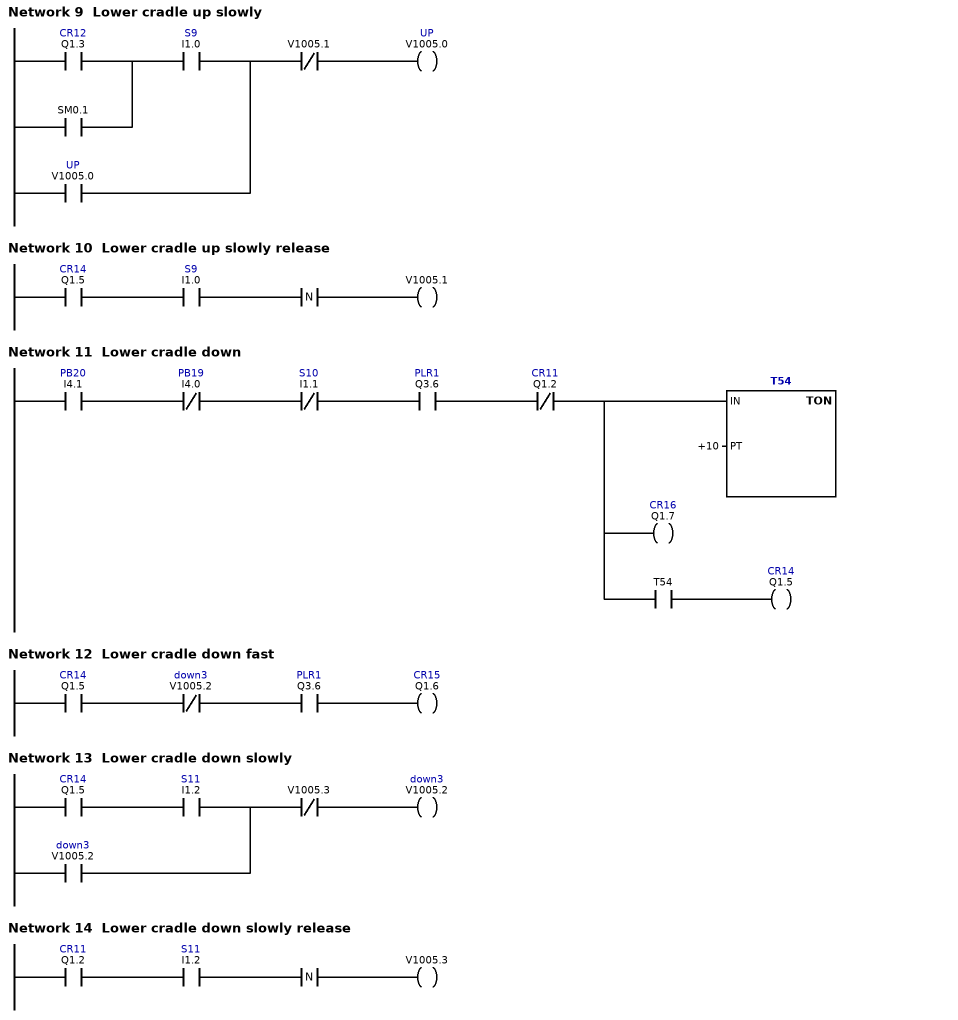
[picture p24: SBR7 networks 9-14]
Network 9 // Lower cradle up slowly
LD     CR12:Q1.3
O      SM0.1
A      S9:I1.0
O      UP:V1005.0
AN     V1005.1
=      UP:V1005.0
Network 10 // Lower cradle up slowly release
LD     CR14:Q1.5
A      S9:I1.0
ED
=      V1005.1
Network 11 // Lower cradle down
LD     PB20:I4.1
AN     PB19:I4.0
AN     S10:I1.1
A      PLR1:Q3.6
AN     CR11:Q1.2
TON    T54, +10
=      CR16:Q1.7
A      T54
=      CR14:Q1.5
Network 12 // Lower cradle down fast
LD     CR14:Q1.5
AN     down3:V1005.2
A      PLR1:Q3.6
=      CR15:Q1.6
Network 13 // Lower cradle down slowly
LD     CR14:Q1.5
A      S11:I1.2
O      down3:V1005.2
AN     V1005.3
=      down3:V1005.2
Network 14 // Lower cradle down slowly release
LD     CR11:Q1.2
A      S11:I1.2
ED
=      V1005.3
END_SUBROUTINE_BLOCK

SUBROUTINE_BLOCK Sheed_lead:SBR8
TITLE= SUBROUTINE COMMENTS
// Press F1 for help and example program 
BEGIN
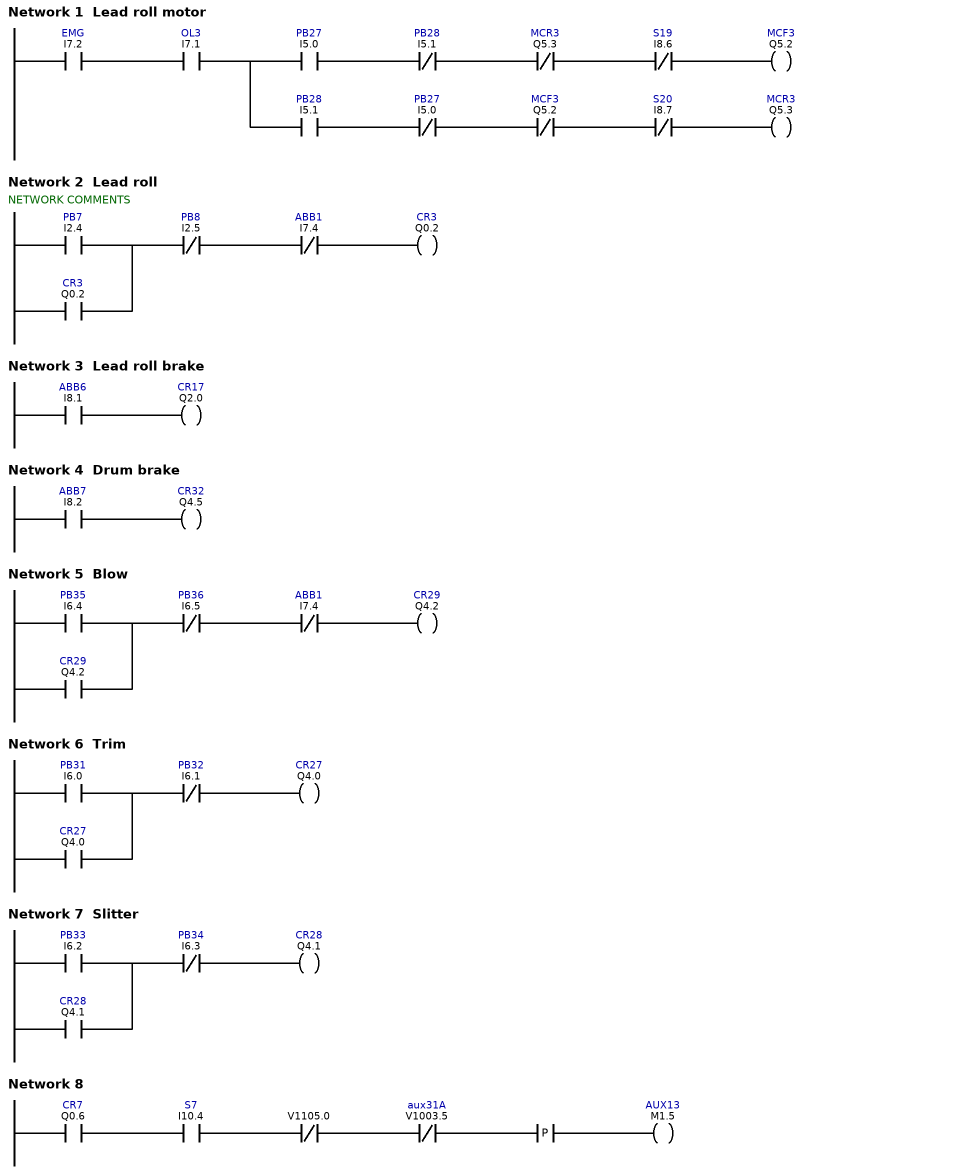
Network 1 // Lead roll motor
LD     EMG:I7.2
A      OL3:I7.1
LPS
A      PB27:I5.0
AN     PB28:I5.1
AN     MCR3:Q5.3
AN     S19:I8.6
=      MCF3:Q5.2
LPP
A      PB28:I5.1
AN     PB27:I5.0
AN     MCF3:Q5.2
AN     S20:I8.7
=      MCR3:Q5.3
Network 2 // Lead roll
//  NETWORK COMMENTS
LD     PB7:I2.4
O      CR3:Q0.2
AN     PB8:I2.5
AN     ABB1:I7.4
=      CR3:Q0.2
Network 3 // Lead roll brake
LD     ABB6:I8.1
=      CR17:Q2.0
Network 4 // Drum brake
LD     ABB7:I8.2
=      CR32:Q4.5
Network 5 // Blow
LD     PB35:I6.4
O      CR29:Q4.2
AN     PB36:I6.5
AN     ABB1:I7.4
=      CR29:Q4.2
Network 6 // Trim 
LD     PB31:I6.0
O      CR27:Q4.0
AN     PB32:I6.1
=      CR27:Q4.0
Network 7 // Slitter
LD     PB33:I6.2
O      CR28:Q4.1
AN     PB34:I6.3
=      CR28:Q4.1
Network 8
LD     CR7:Q0.6
A      S7:I10.4
AN     V1105.0
AN     aux31A:V1003.5
EU
=      AUX13:M1.5
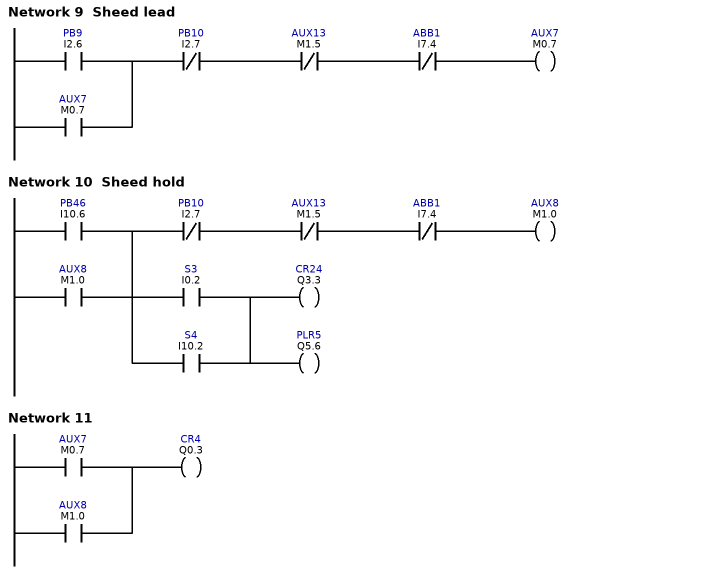
Network 9 // Sheed lead
LD     PB9:I2.6
O      AUX7:M0.7
AN     PB10:I2.7
AN     AUX13:M1.5
AN     ABB1:I7.4
=      AUX7:M0.7
Network 10 // Sheed hold
LD     PB46:I10.6
O      AUX8:M1.0
LPS
AN     PB10:I2.7
AN     AUX13:M1.5
AN     ABB1:I7.4
=      AUX8:M1.0
LPP
LD     S3:I0.2
O      S4:I10.2
ALD
=      CR24:Q3.3
=      PLR5:Q5.6
Network 11
LD     AUX7:M0.7
O      AUX8:M1.0
=      CR4:Q0.3
END_SUBROUTINE_BLOCK

SUBROUTINE_BLOCK Core_Chuck:SBR9
TITLE= 
// SUBROUTINE COMMENTS
// Press F1 for help and example program
//  
BEGIN
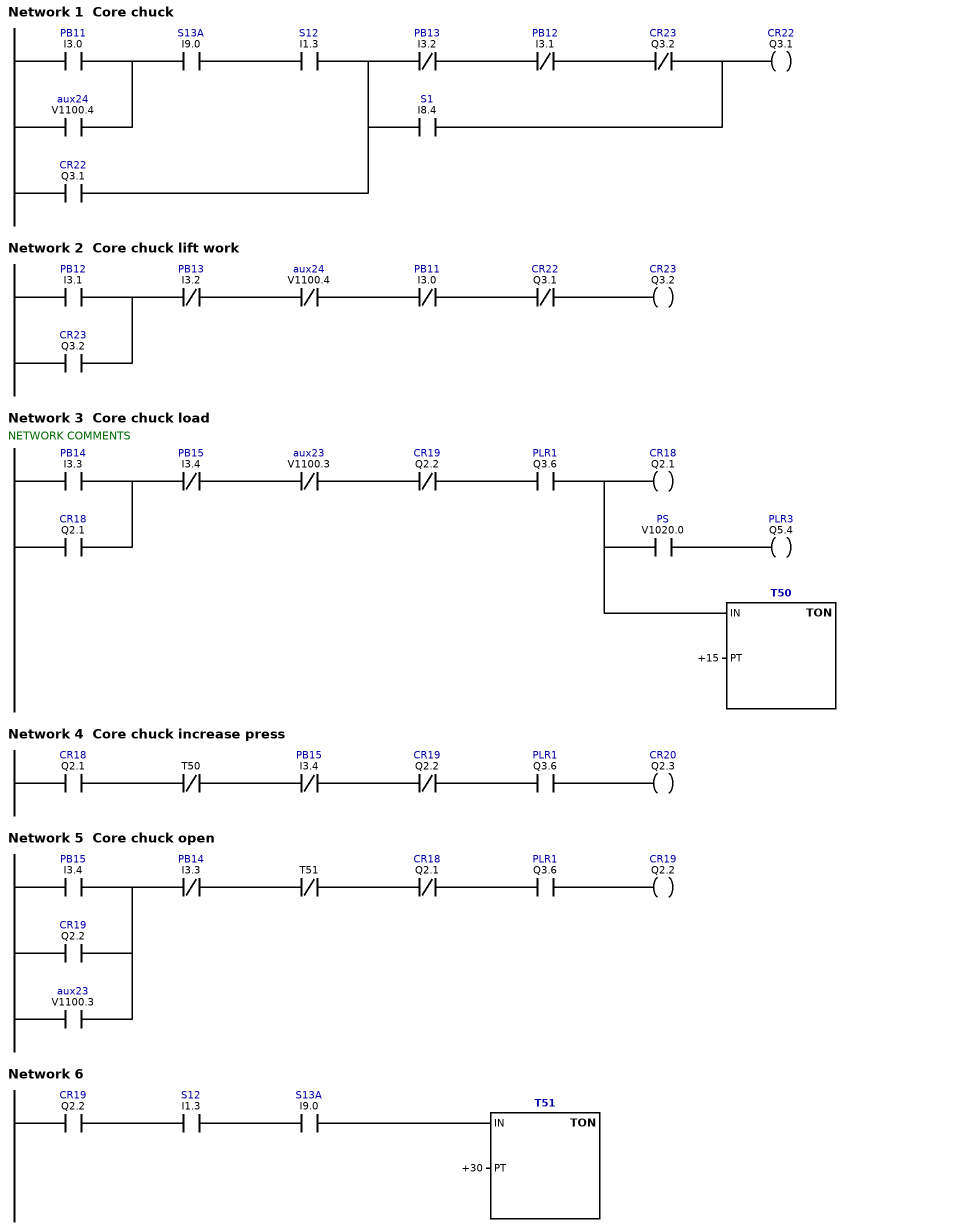
Network 1 // Core chuck
// 
// 
LD     PB11:I3.0
O      aux24:V1100.4
A      S13A:I9.0
A      S12:I1.3
O      CR22:Q3.1
LDN    PB13:I3.2
AN     PB12:I3.1
AN     CR23:Q3.2
O      S1:I8.4
ALD
=      CR22:Q3.1
Network 2 // Core chuck lift work
// 
// 
LD     PB12:I3.1
O      CR23:Q3.2
AN     PB13:I3.2
AN     aux24:V1100.4
AN     PB11:I3.0
AN     CR22:Q3.1
=      CR23:Q3.2
Network 3 // Core chuck load
//  NETWORK COMMENTS
LD     PB14:I3.3
O      CR18:Q2.1
AN     PB15:I3.4
AN     aux23:V1100.3
AN     CR19:Q2.2
A      PLR1:Q3.6
LPS
=      CR18:Q2.1
A      PS:V1020.0
=      PLR3:Q5.4
LPP
TON    T50, +15
Network 4 // Core chuck increase press
LD     CR18:Q2.1
AN     T50
AN     PB15:I3.4
AN     CR19:Q2.2
A      PLR1:Q3.6
=      CR20:Q2.3
Network 5 // Core chuck open
LD     PB15:I3.4
O      CR19:Q2.2
O      aux23:V1100.3
AN     PB14:I3.3
AN     T51
AN     CR18:Q2.1
A      PLR1:Q3.6
=      CR19:Q2.2
Network 6
LD     CR19:Q2.2
A      S12:I1.3
A      S13A:I9.0
TON    T51, +30
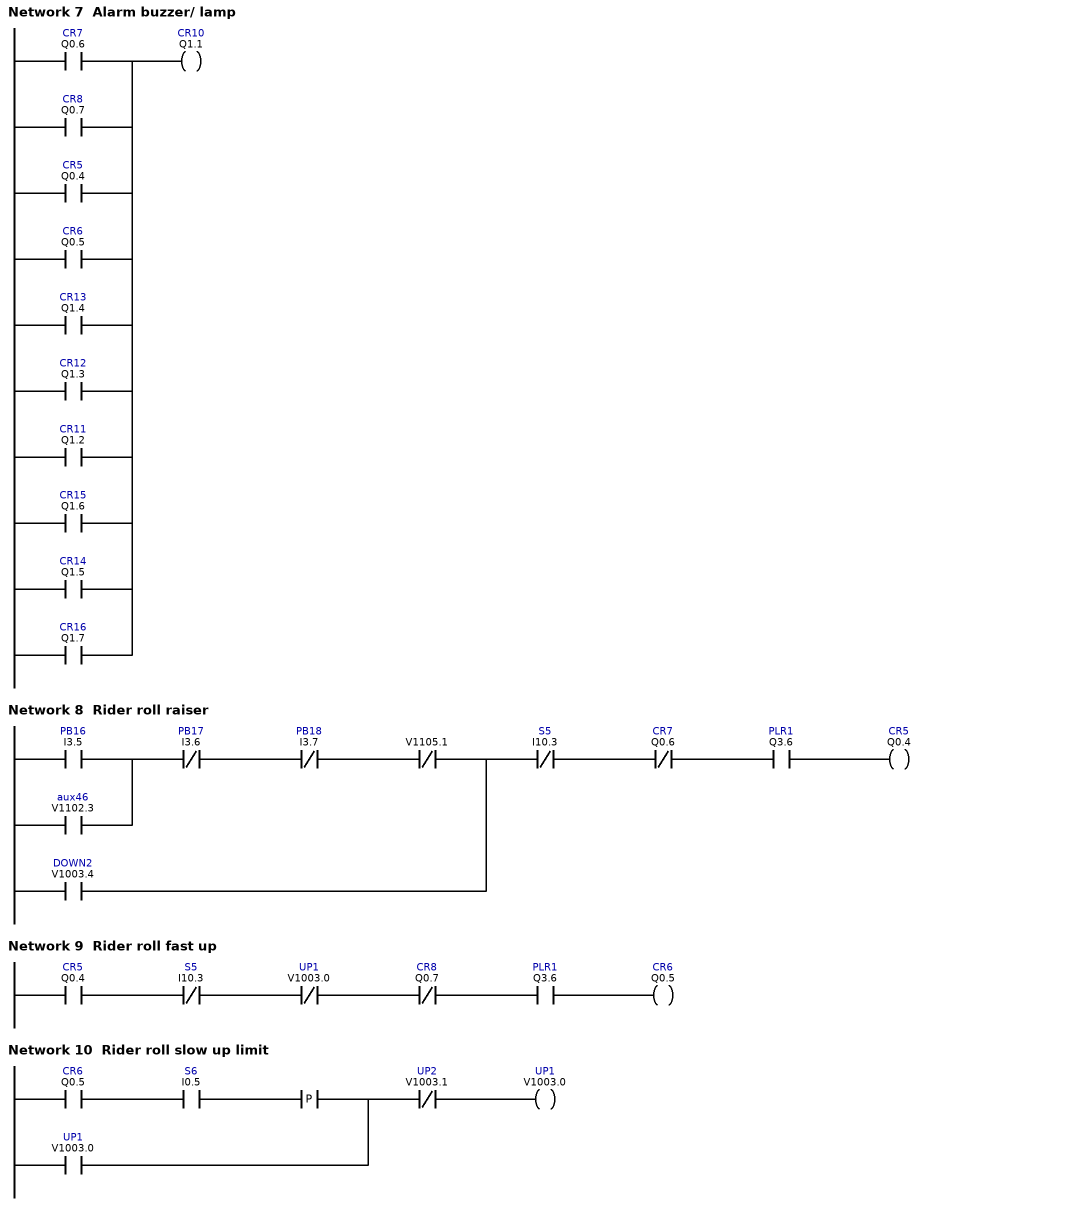
Network 7 // Alarm buzzer/ lamp
LD     CR7:Q0.6
O      CR8:Q0.7
O      CR5:Q0.4
O      CR6:Q0.5
O      CR13:Q1.4
O      CR12:Q1.3
O      CR11:Q1.2
O      CR15:Q1.6
O      CR14:Q1.5
O      CR16:Q1.7
=      CR10:Q1.1
Network 8 // Rider roll raiser
LD     PB16:I3.5
O      aux46:V1102.3
AN     PB17:I3.6
AN     PB18:I3.7
AN     V1105.1
O      DOWN2:V1003.4
AN     S5:I10.3
AN     CR7:Q0.6
A      PLR1:Q3.6
=      CR5:Q0.4
Network 9 // Rider roll fast up
LD     CR5:Q0.4
AN     S5:I10.3
AN     UP1:V1003.0
AN     CR8:Q0.7
A      PLR1:Q3.6
=      CR6:Q0.5
Network 10 // Rider roll slow up limit
LD     CR6:Q0.5
A      S6:I0.5
EU
O      UP1:V1003.0
AN     UP2:V1003.1
=      UP1:V1003.0
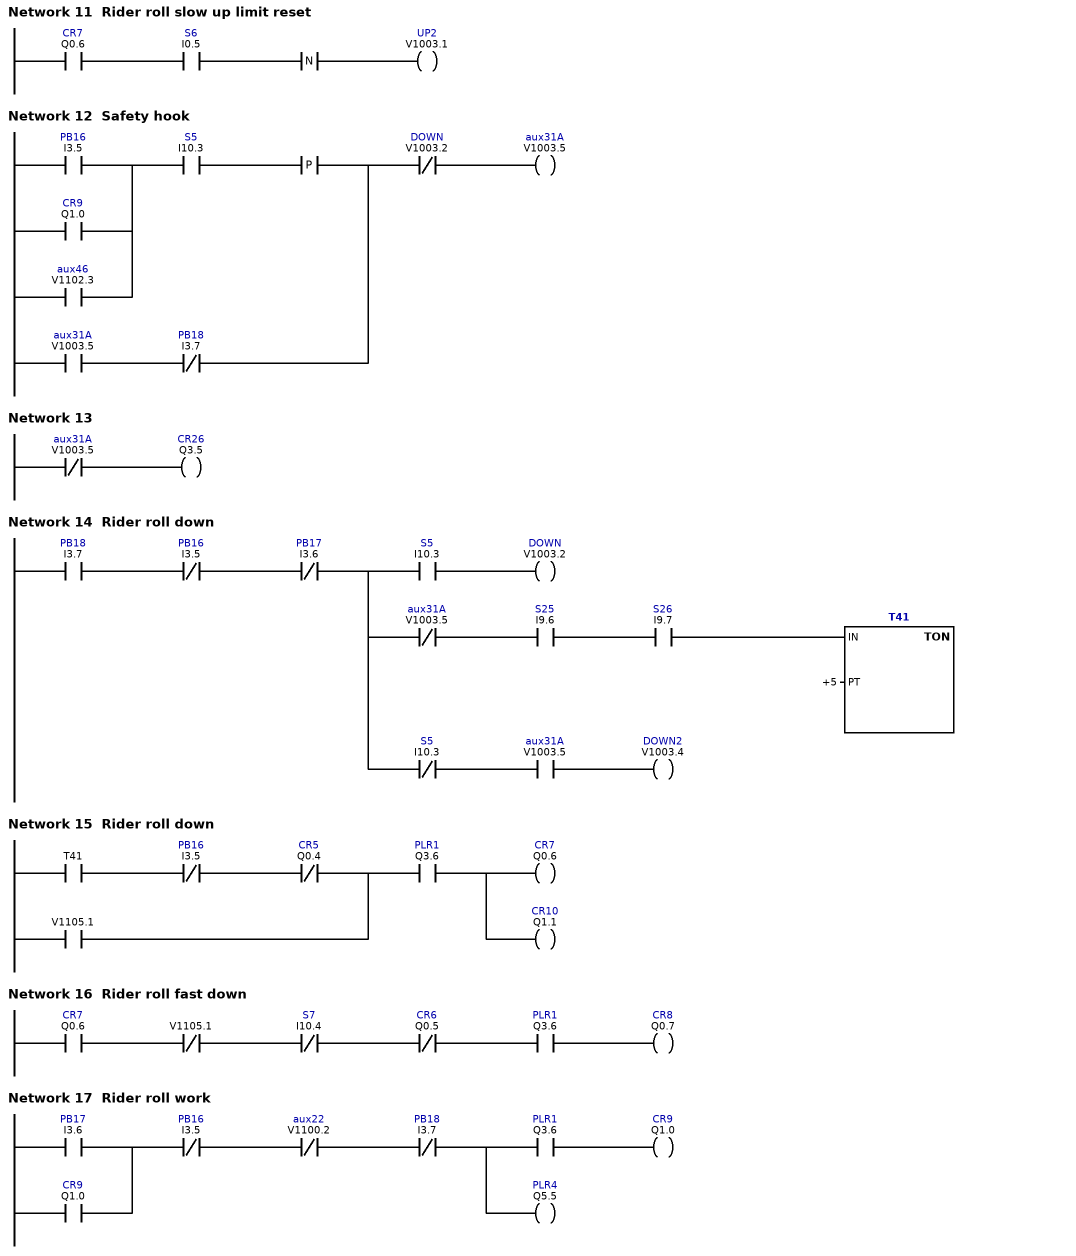
Network 11 // Rider roll slow up limit reset
LD     CR7:Q0.6
A      S6:I0.5
ED
=      UP2:V1003.1
Network 12 // Safety hook
LD     PB16:I3.5
O      CR9:Q1.0
O      aux46:V1102.3
A      S5:I10.3
EU
LD     aux31A:V1003.5
AN     PB18:I3.7
OLD
AN     DOWN:V1003.2
=      aux31A:V1003.5
Network 13
LDN    aux31A:V1003.5
=      CR26:Q3.5
Network 14 // Rider roll down
LD     PB18:I3.7
AN     PB16:I3.5
AN     PB17:I3.6
LPS
A      S5:I10.3
=      DOWN:V1003.2
LRD
AN     aux31A:V1003.5
A      S25:I9.6
A      S26:I9.7
TON    T41, +5
LPP
AN     S5:I10.3
A      aux31A:V1003.5
=      DOWN2:V1003.4
Network 15 // Rider roll down
LD     T41
AN     PB16:I3.5
AN     CR5:Q0.4
O      V1105.1
A      PLR1:Q3.6
=      CR7:Q0.6
=      CR10:Q1.1
Network 16 // Rider roll fast down
LD     CR7:Q0.6
AN     V1105.1
AN     S7:I10.4
AN     CR6:Q0.5
A      PLR1:Q3.6
=      CR8:Q0.7
Network 17 // Rider roll work
LD     PB17:I3.6
O      CR9:Q1.0
AN     PB16:I3.5
AN     aux22:V1100.2
AN     PB18:I3.7
LPS
A      PLR1:Q3.6
=      CR9:Q1.0
LPP
=      PLR4:Q5.5
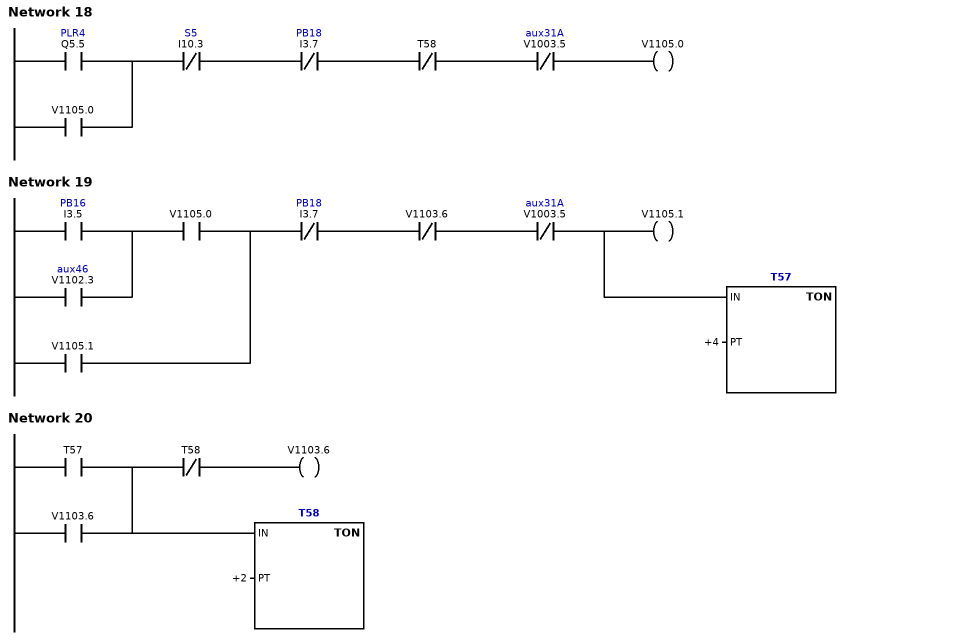
Network 18
LD     PLR4:Q5.5
O      V1105.0
AN     S5:I10.3
AN     PB18:I3.7
AN     T58
AN     aux31A:V1003.5
=      V1105.0
Network 19
LD     PB16:I3.5
O      aux46:V1102.3
A      V1105.0
O      V1105.1
AN     PB18:I3.7
AN     V1103.6
AN     aux31A:V1003.5
=      V1105.1
TON    T57, +4
Network 20
LD     T57
O      V1103.6
LPS
AN     T58
=      V1103.6
LPP
TON    T58, +2
END_SUBROUTINE_BLOCK

SUBROUTINE_BLOCK Value_1:SBR10
TITLE= SUBROUTINE COMMENTS
// Press F1 for help and example program 
VAR_INPUT
d1:REAL;	// LD0 
H:REAL;	// LD4 
END_VAR
VAR_OUTPUT
D:REAL;	// LD8 
END_VAR
VAR
TEMP1:REAL;	// LD12 
TEMP2:REAL;	// LD16 
TEMP3:REAL;	// LD20 
TEMP4:REAL;	// LD24 
TEMP5:REAL;	// LD28 
TEMP6:REAL;	// LD32 
TEMP7:REAL;	// LD36 
TEMP8:REAL;	// LD40 
TEMP9:REAL;	// LD44 
TEMP10:REAL;	// LD48 
TEMP11:REAL;	// LD52 
END_VAR
BEGIN
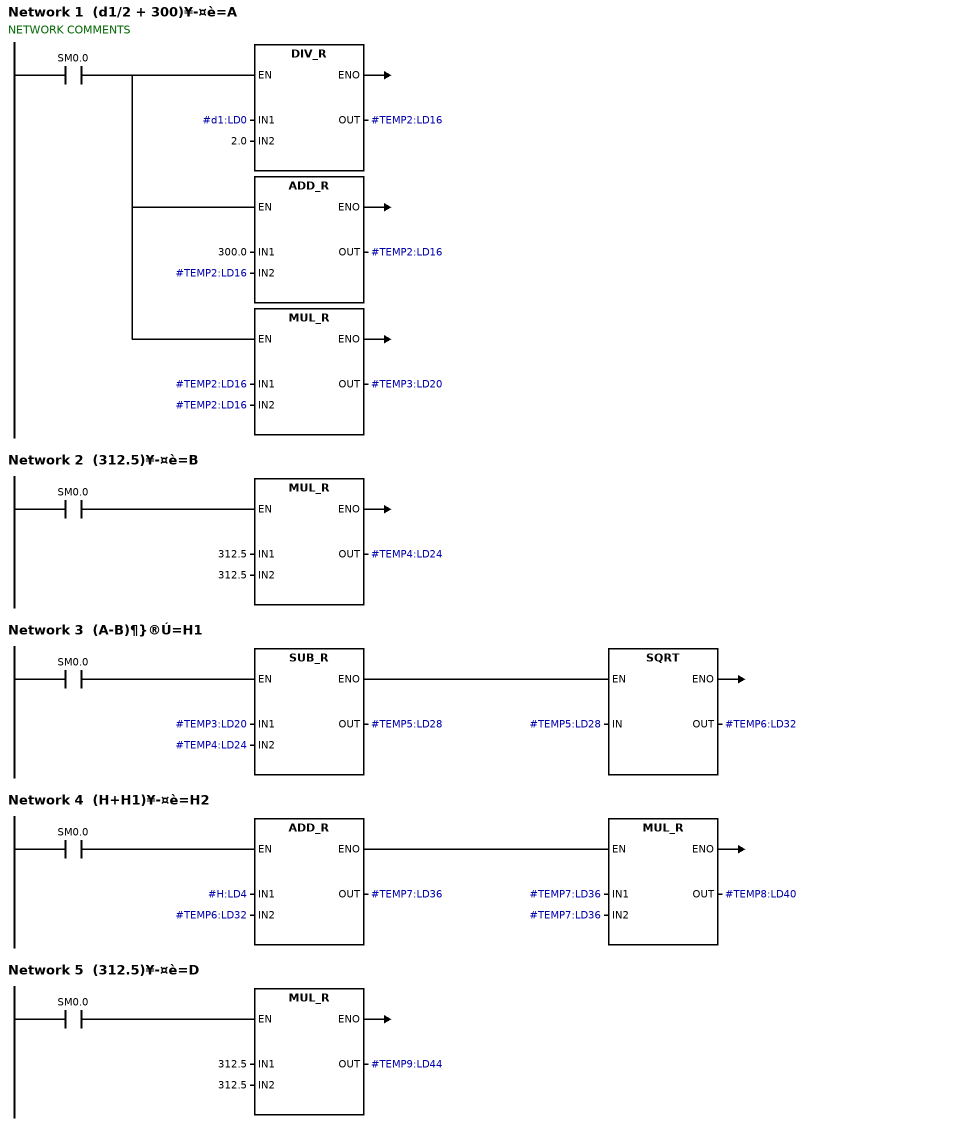
Network 1 // (d1/2 + 300)平方=A
//  NETWORK COMMENTS
LD     SM0.0
MOVR   #d1:LD0, #TEMP2:LD16
/R     2.0, #TEMP2:LD16
+R     300.0, #TEMP2:LD16
MOVR   #TEMP2:LD16, #TEMP3:LD20
*R     #TEMP2:LD16, #TEMP3:LD20
Network 2 // (312.5)平方=B
LD     SM0.0
MOVR   312.5, #TEMP4:LD24
*R     312.5, #TEMP4:LD24
Network 3 // (A-B)開根=H1
LD     SM0.0
MOVR   #TEMP3:LD20, #TEMP5:LD28
AENO
-R     #TEMP4:LD24, #TEMP5:LD28
AENO
SQRT   #TEMP5:LD28, #TEMP6:LD32
Network 4 // (H+H1)平方=H2
LD     SM0.0
MOVR   #H:LD4, #TEMP7:LD36
AENO
+R     #TEMP6:LD32, #TEMP7:LD36
AENO
MOVR   #TEMP7:LD36, #TEMP8:LD40
*R     #TEMP7:LD36, #TEMP8:LD40
Network 5 // (312.5)平方=D
LD     SM0.0
MOVR   312.5, #TEMP9:LD44
*R     312.5, #TEMP9:LD44
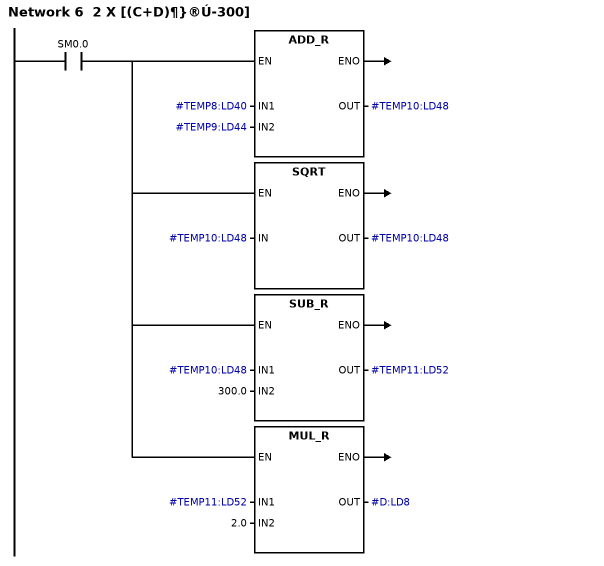
Network 6 // 2 X [(C+D)開根-300]
LD     SM0.0
MOVR   #TEMP8:LD40, #TEMP10:LD48
+R     #TEMP9:LD44, #TEMP10:LD48
SQRT   #TEMP10:LD48, #TEMP10:LD48
MOVR   #TEMP10:LD48, #TEMP11:LD52
-R     300.0, #TEMP11:LD52
MOVR   #TEMP11:LD52, #D:LD8
*R     2.0, #D:LD8
Network 8 // NETWORK TITLE (single line)
//  
// NETWORK COMMENTS
//  
// 
END_SUBROUTINE_BLOCK

SUBROUTINE_BLOCK TOSHIBA_DO:SBR11
TITLE= SUBROUTINE COMMENTS
// Press F1 for help and example program 
BEGIN
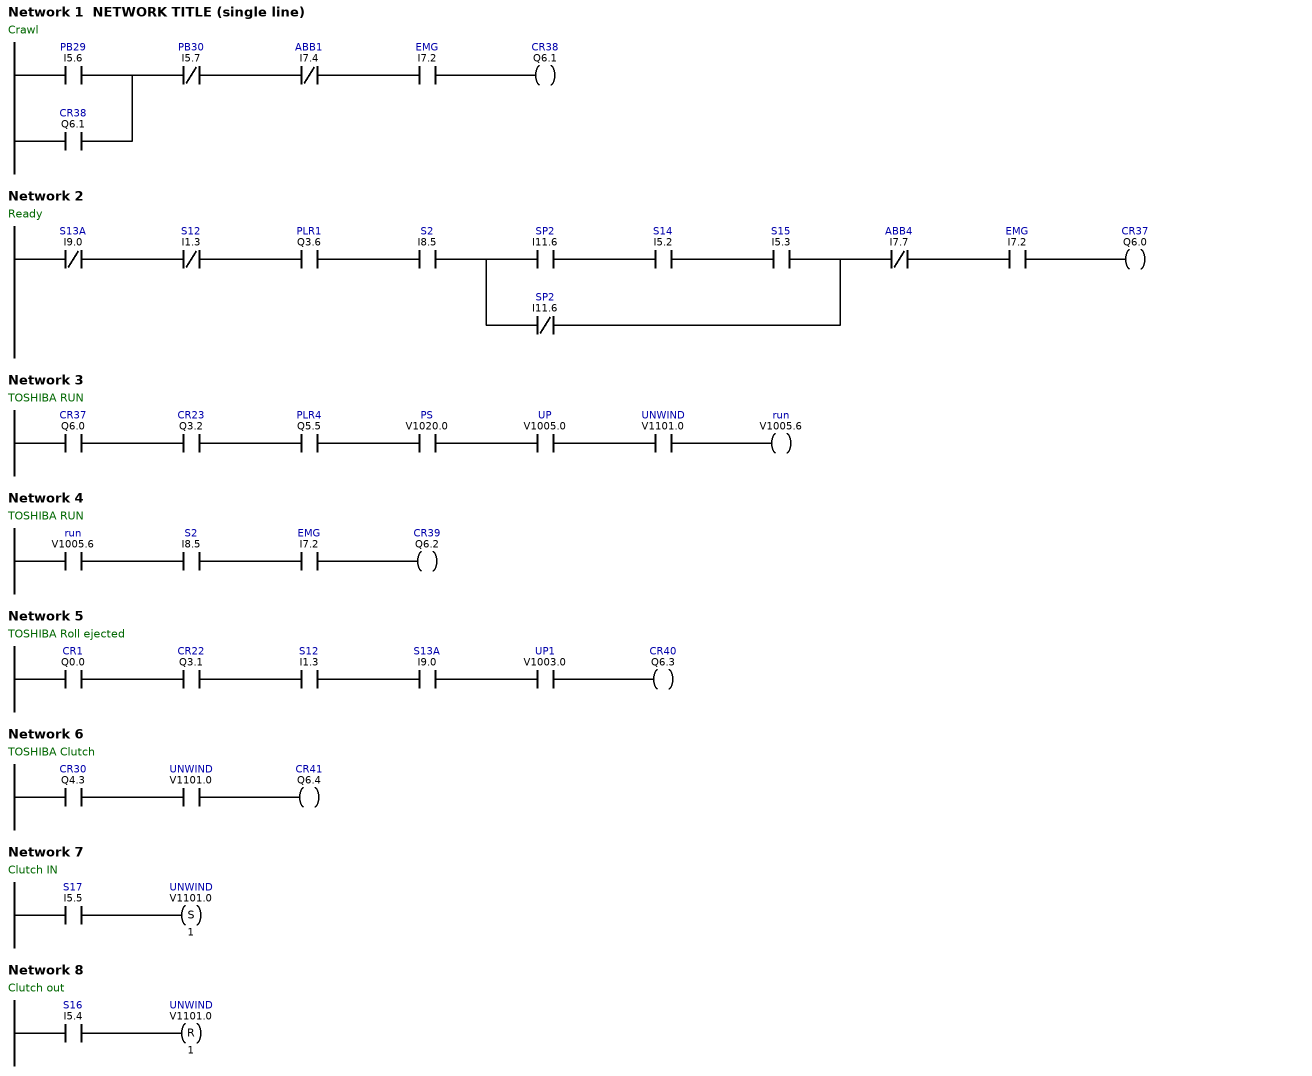
Network 1 // NETWORK TITLE (single line)
// Crawl
LD     PB29:I5.6
O      CR38:Q6.1
AN     PB30:I5.7
AN     ABB1:I7.4
A      EMG:I7.2
=      CR38:Q6.1
Network 2
// Ready
LDN    S13A:I9.0
AN     S12:I1.3
A      PLR1:Q3.6
A      S2:I8.5
LD     SP2:I11.6
A      S14:I5.2
A      S15:I5.3
ON     SP2:I11.6
ALD
AN     ABB4:I7.7
A      EMG:I7.2
=      CR37:Q6.0
Network 3
// TOSHIBA RUN
LD     CR37:Q6.0
A      CR23:Q3.2
A      PLR4:Q5.5
A      PS:V1020.0
A      UP:V1005.0
A      UNWIND:V1101.0
=      run:V1005.6
Network 4
// TOSHIBA RUN
LD     run:V1005.6
A      S2:I8.5
A      EMG:I7.2
=      CR39:Q6.2
Network 5
// TOSHIBA Roll ejected
LD     CR1:Q0.0
A      CR22:Q3.1
A      S12:I1.3
A      S13A:I9.0
A      UP1:V1003.0
=      CR40:Q6.3
Network 6
// TOSHIBA Clutch
LD     CR30:Q4.3
A      UNWIND:V1101.0
=      CR41:Q6.4
Network 7
// Clutch IN
LD     S17:I5.5
S      UNWIND:V1101.0, 1
Network 8
// Clutch out
LD     S16:I5.4
R      UNWIND:V1101.0, 1
END_SUBROUTINE_BLOCK

SUBROUTINE_BLOCK Auto_Roll_Eiector:SBR12
TITLE=SUBROUTINE COMMENTS
BEGIN
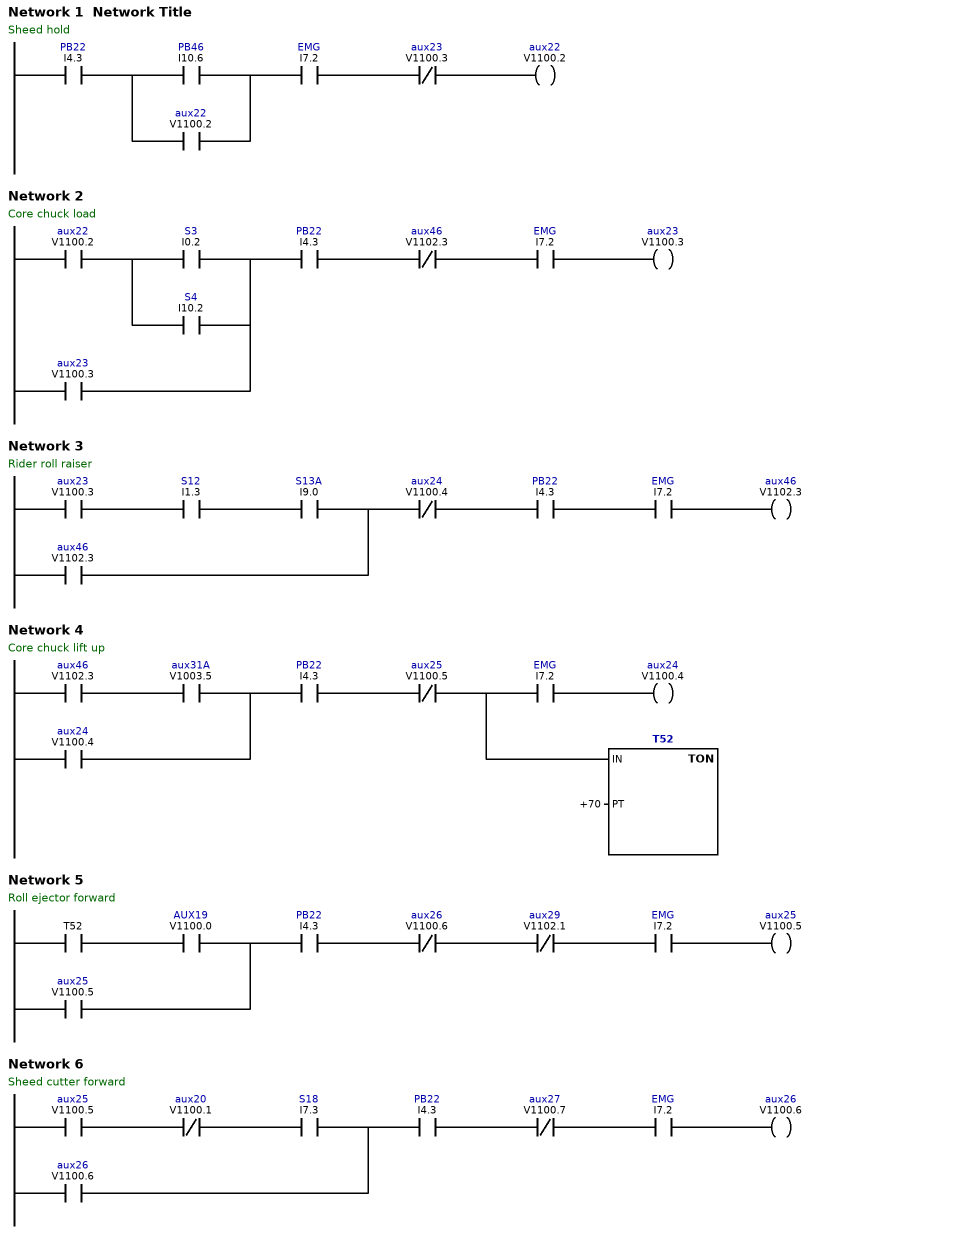
Network 1 // Network Title
// Sheed hold
LD     PB22:I4.3
LD     PB46:I10.6
O      aux22:V1100.2
ALD
A      EMG:I7.2
AN     aux23:V1100.3
=      aux22:V1100.2
Network 2
// Core chuck load
LD     aux22:V1100.2
LD     S3:I0.2
O      S4:I10.2
ALD
O      aux23:V1100.3
A      PB22:I4.3
AN     aux46:V1102.3
A      EMG:I7.2
=      aux23:V1100.3
Network 3
// Rider roll raiser
LD     aux23:V1100.3
A      S12:I1.3
A      S13A:I9.0
O      aux46:V1102.3
AN     aux24:V1100.4
A      PB22:I4.3
A      EMG:I7.2
=      aux46:V1102.3
Network 4
// Core chuck lift up
LD     aux46:V1102.3
A      aux31A:V1003.5
O      aux24:V1100.4
A      PB22:I4.3
AN     aux25:V1100.5
LPS
A      EMG:I7.2
=      aux24:V1100.4
LPP
TON    T52, +70
Network 5
// Roll ejector forward
LD     T52
A      AUX19:V1100.0
O      aux25:V1100.5
A      PB22:I4.3
AN     aux26:V1100.6
AN     aux29:V1102.1
A      EMG:I7.2
=      aux25:V1100.5
Network 6
// Sheed cutter forward
LD     aux25:V1100.5
AN     aux20:V1100.1
A      S18:I7.3
O      aux26:V1100.6
A      PB22:I4.3
AN     aux27:V1100.7
A      EMG:I7.2
=      aux26:V1100.6
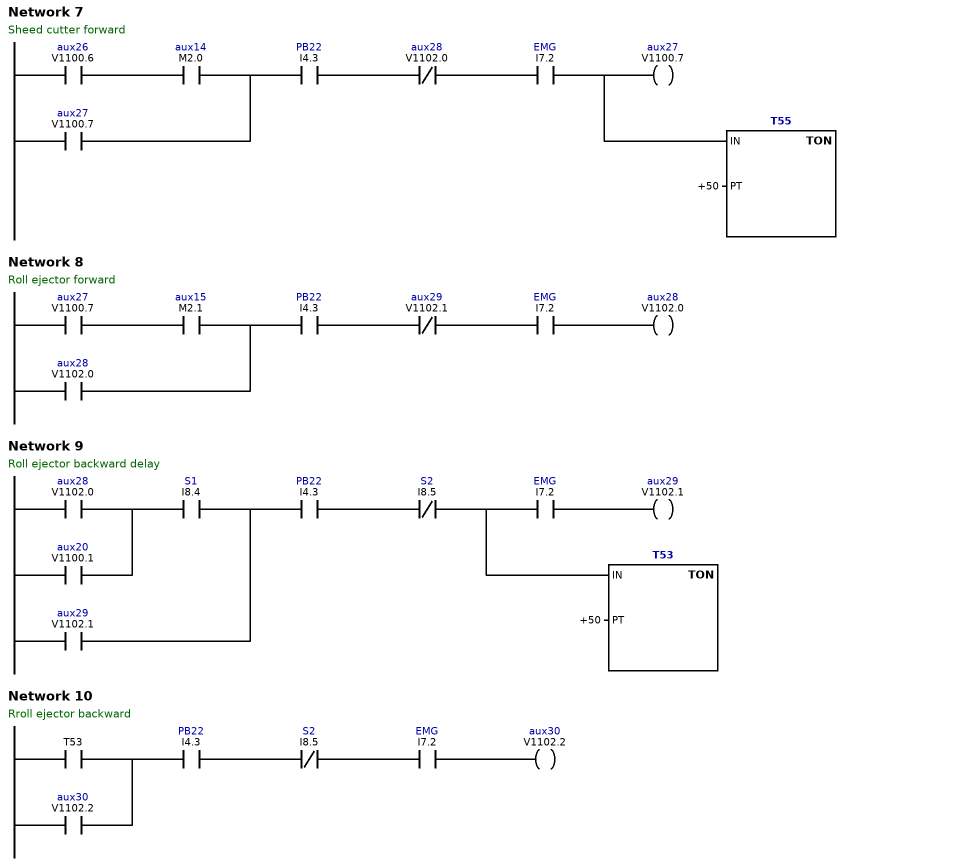
Network 7
// Sheed cutter forward
LD     aux26:V1100.6
A      aux14:M2.0
O      aux27:V1100.7
A      PB22:I4.3
AN     aux28:V1102.0
A      EMG:I7.2
=      aux27:V1100.7
TON    T55, +50
Network 8
// Roll ejector forward
LD     aux27:V1100.7
A      aux15:M2.1
O      aux28:V1102.0
A      PB22:I4.3
AN     aux29:V1102.1
A      EMG:I7.2
=      aux28:V1102.0
Network 9
// Roll ejector backward delay
LD     aux28:V1102.0
O      aux20:V1100.1
A      S1:I8.4
O      aux29:V1102.1
A      PB22:I4.3
AN     S2:I8.5
LPS
A      EMG:I7.2
=      aux29:V1102.1
LPP
TON    T53, +50
Network 10
// Rroll ejector backward
LD     T53
O      aux30:V1102.2
A      PB22:I4.3
AN     S2:I8.5
A      EMG:I7.2
=      aux30:V1102.2
END_SUBROUTINE_BLOCK

SUBROUTINE_BLOCK TOSHIBA_Diameter_AO:SBR13
TITLE=
VAR_INPUT
temp0:REAL;	// LD0 
END_VAR
VAR_OUTPUT
temp6:REAL;	// LD4 
END_VAR
VAR
temp1:REAL;	// LD8 
temp2:REAL;	// LD12 
temp3:REAL;	// LD16 
END_VAR
BEGIN
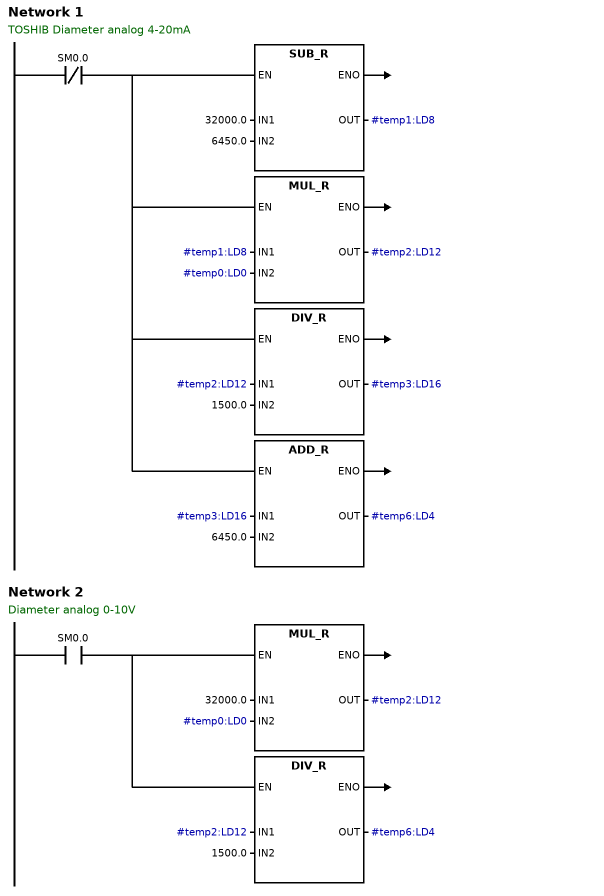
Network 1
// TOSHIB Diameter analog 4-20mA
LDN    SM0.0
MOVR   32000.0, #temp1:LD8
-R     6450.0, #temp1:LD8
MOVR   #temp1:LD8, #temp2:LD12
*R     #temp0:LD0, #temp2:LD12
MOVR   #temp2:LD12, #temp3:LD16
/R     1500.0, #temp3:LD16
MOVR   #temp3:LD16, #temp6:LD4
+R     6450.0, #temp6:LD4
Network 2
// Diameter analog 0-10V
LD     SM0.0
MOVR   32000.0, #temp2:LD12
*R     #temp0:LD0, #temp2:LD12
MOVR   #temp2:LD12, #temp6:LD4
/R     1500.0, #temp6:LD4
END_SUBROUTINE_BLOCK

SUBROUTINE_BLOCK System_fault:SBR14
TITLE=
BEGIN
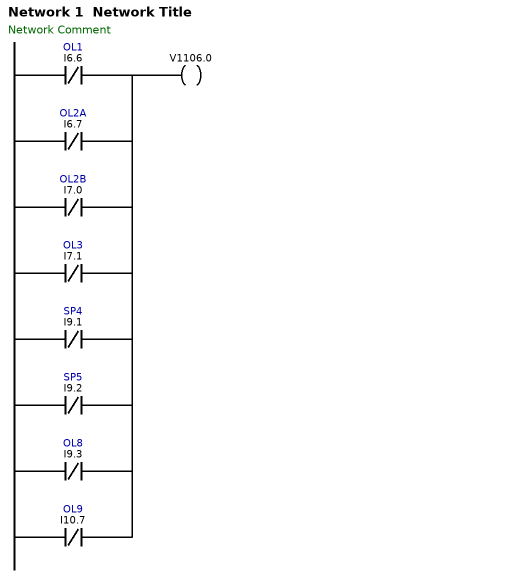
Network 1 // Network Title
// Network Comment
LDN    OL1:I6.6
ON     OL2A:I6.7
ON     OL2B:I7.0
ON     OL3:I7.1
ON     SP4:I9.1
ON     SP5:I9.2
ON     OL8:I9.3
ON     OL9:I10.7
=      V1106.0
END_SUBROUTINE_BLOCK
